// TIA Portal V16 export
// export: Created 2024-01-13T18:16:19.9688211Z, ExportSetting WithDefaults, DisplayName Totally Integrated Automation Portal, DisplayVersion V16, DisplayName TIA Portal Version Control Interface, DisplayVersion V16, DisplayName TIA Portal Openness, DisplayVersion V16, DisplayName STEP 7 Professional, DisplayVersion V16, DisplayName STEP 7 Safety, DisplayVersion V16, DisplayName WinCC Professional, DisplayVersion V16
VAR_GLOBAL   // PLC tag table "Default tag table"
   Tag_1 AT %MW0 : Word;
   Tag_2 AT %M2.0 : Bool;
   Tag_3 AT %M2.1 : Bool;
   Tag_4 AT %M2.2 : Bool;
   Tag_5 AT %M2.3 : Bool;
   Tag_6 AT %M2.4 : Bool;
   Tag_7 AT %M2.5 : Bool;
   Tag_8 AT %M2.6 : Bool;
   Tag_9 AT %M2.7 : Bool;
   Tag_10 AT %M3.0 : Bool;
   Tag_11 AT %M3.1 : Bool;
   Tag_12 AT %M3.2 : Bool;
   Tag_13 AT %M3.3 : Bool;
   Tag_14 AT %M3.4 : Bool;
END_VAR
